{attribute 'pack_mode' := '1'}
TYPE ST_OpcUa_PointBase :
STRUCT
  TimeStamp : ULINT;
  ErrorCode : UDINT;
END_STRUCT
END_TYPE

(* stored: Version 1.1.0.1, ProductVersion 3.1.4024.9
   DUT ST_OpcUa_PointBase: Id {47451af4-e2bb-4712-820e-db43d0179042} *)
